FUNCTION_BLOCK UNIT_Blikkenvullijn IMPLEMENTS  ITF_Blikkenvullijn
VAR
	EM_Can_Supply 		: FB_Can_Supply;
	EM_Filling			: FB_Machine_PackML;
	EM_Check_Weigher	: FB_Machine_PackML;
	EM_Labeller			: FB_Machine_PackML;
	EM_Turning			: FB_Machine_PackML;
	EM_Stamp			: FB_Machine_PackML;
	EM_Seal_Shrink		: FB_Machine_PackML;
END_VAR

(*
$$$$$$$$\                                                                   $$\       $$$$$$$$\                     $$\                                         $$\                     
$$  _____|                                                                  $$ |      $$  _____|                    \__|                                        \__|                    
$$ |   $$$$$$\   $$$$$$\  $$$$$$$\  $$\  $$\  $$\  $$$$$$\   $$$$$$\   $$$$$$$ |      $$ |      $$$$$$$\   $$$$$$\  $$\ $$$$$$$\   $$$$$$\   $$$$$$\   $$$$$$\  $$\ $$$$$$$\   $$$$$$\  
$$$$$\ \____$$\ $$  __$$\ $$  __$$\ $$ | $$ | $$ |$$  __$$\ $$  __$$\ $$  __$$ |      $$$$$\    $$  __$$\ $$  __$$\ $$ |$$  __$$\ $$  __$$\ $$  __$$\ $$  __$$\ $$ |$$  __$$\ $$  __$$\ 
$$  __|$$$$$$$ |$$ |  \__|$$ |  $$ |$$ | $$ | $$ |$$ /  $$ |$$ /  $$ |$$ /  $$ |      $$  __|   $$ |  $$ |$$ /  $$ |$$ |$$ |  $$ |$$$$$$$$ |$$$$$$$$ |$$ |  \__|$$ |$$ |  $$ |$$ /  $$ |
$$ |  $$  __$$ |$$ |      $$ |  $$ |$$ | $$ | $$ |$$ |  $$ |$$ |  $$ |$$ |  $$ |      $$ |      $$ |  $$ |$$ |  $$ |$$ |$$ |  $$ |$$   ____|$$   ____|$$ |      $$ |$$ |  $$ |$$ |  $$ |
$$ |  \$$$$$$$ |$$ |      $$ |  $$ |\$$$$$\$$$$  |\$$$$$$  |\$$$$$$  |\$$$$$$$ |      $$$$$$$$\ $$ |  $$ |\$$$$$$$ |$$ |$$ |  $$ |\$$$$$$$\ \$$$$$$$\ $$ |      $$ |$$ |  $$ |\$$$$$$$ |
\__|   \_______|\__|      \__|  \__| \_____\____/  \______/  \______/  \_______|      \________|\__|  \__| \____$$ |\__|\__|  \__| \_______| \_______|\__|      \__|\__|  \__| \____$$ |
                                                                                                          $$\   $$ |                                                          $$\   $$ |
                                                                                                          \$$$$$$  |                                                          \$$$$$$  |
                                                                                                           \______/                                                            \______/ 
*)

//**************************INITIATE**************************//
//*****************************EM*****************************//
//*************************BlackBoxes*************************//
EM_Filling();
EM_Check_Weigher();
EM_Labeller();
EM_Turning();
EM_Stamp();
EM_Seal_Shrink();
//*************************Custommade*************************//
EM_Can_Supply();

METHOD FB_init : BOOL
VAR_INPUT
	bInitRetains : BOOL; // if TRUE, the retain variables are initialized (warm start / cold start)
	bInCopyCode : BOOL;  // if TRUE, the instance afterwards gets moved into the copy code (online change)
END_VAR
//*****************************INITIATE*****************************//
EM_Can_Supply.FB_init(0,0);
EM_Filling.FB_init(0,0);
EM_Check_Weigher.FB_init(0,0);
EM_Labeller.FB_init(0,0);
EM_Turning.FB_init(0,0);
EM_Stamp.FB_init(0,0);
EM_Seal_Shrink.FB_init(0,0);
END_METHOD

END_FUNCTION_BLOCK

(* stored: Version 1.1.0.1, ProductVersion 3.1.4024.12
   POU UNIT_Blikkenvullijn: Id {2692377b-29af-456d-aace-ede4a94c185d}, SpecialFunc None
   Method FB_init: Id {e016cb9e-71c8-4e78-924d-1e46be021f7d} *)
